GLOBALCONSTANTS ISOUSERHOME_e (* CF / User network location *)
  (* Standard: 61499-1 *)
  (* Version 1.0, 2025-10-18, franz *)
  PACKAGE isobus::pgn;
  VAR_GLOBAL CONSTANT
    intern : SINT := 0;
    network : SINT := 1;
    thisMember : SINT := 2;
    notdef : SINT := -1;
  END_VAR
END_GLOBALCONSTANTS
